{attribute 'GeneratedUsingTerminal: EL3122--0000'}
{attribute addProperty BoxType "EL3122--0000"}
{attribute addProperty Id "EtcSlaveTerminalBaseChannel_1AT %I*Channel_7539AA333Channel_2AT %I*Channel_7539AA333WcStateAT %I*WcState_9091E0EB2InfoDataAT %I*InfoData_32EB74EA10"}
{attribute addProperty CRC "577888235"}
{attribute addProperty Size "18"}
TYPE EL3122_2271DFEB EXTENDS EtcSlaveTerminalBase :
STRUCT
	{attribute addProperty Name "Channel_1"}
	Channel_1 : Channel_7539AA33;
	{attribute addProperty Name "Channel_2"}
	Channel_2 : Channel_7539AA33;
	{attribute addProperty Name "WcState"}
	WcState : WcState_9091E0EB;
	{attribute addProperty Name "InfoData"}
	InfoData : InfoData_32EB74EA;
END_STRUCT
END_TYPE

(* stored: Version 1.2.0.0, ProductVersion 3.1.4024.9
   DUT EL3122_2271DFEB: Id {7740b28b-2c10-4064-9c65-487bee69738f} *)
